FUNCTION UpdateEventTimeWithSystemTime  
VAR_INPUT
	stEvent :REFERENCE TO ST_Event;
END_VAR
	
VAR
	fbLocalSystemTime	:FB_LocalSystemTime := (bEnable := TRUE);
	fbGETSYSTEMTIME 	:GETSYSTEMTIME;
	stT_FILETIME		:T_FILETIME;
END_VAR



stEvent.dtTimeStamp:= SF.systemTime;

END_FUNCTION

(* stored: Version 1.1.0.1, ProductVersion 3.1.4026.18
   POU UpdateEventTimeWithSystemTime: Id {68eb53f8-bbbd-4b65-9c4f-3dd21164492c}, SpecialFunc None *)
